FUNCTION_BLOCK T_ReleaseHandle IMPLEMENTS I_Executable
VAR
   logger : I_Logger;
	_symbolHandle : ST_SymbolHandle;
	write : T_AdsWrite;
END_VAR
VAR CONSTANT
   LOG_DEBUG : DWORD := 0;
   LOG_INFO : DWORD := ADSLOG_MSGTYPE_HINT;
   LOG_WARNING : DWORD := ADSLOG_MSGTYPE_WARN;
   LOG_ERROR : DWORD := ADSLOG_MSGTYPE_ERROR;
END_VAR

write();

PROPERTY Busy : BOOL
GET
Busy := write.Busy;
END_GET
END_PROPERTY

PROPERTY Done : BOOL
GET
Done := write.Done;
END_GET
END_PROPERTY

PROPERTY Error : BOOL
GET
Error := write.Error;
END_GET
END_PROPERTY

METHOD PRIVATE ToLog
VAR_INPUT
	Msg : STRING(255);
	LogLevel : DWORD; // generic level, can be mapped to logging framework
END_VAR
IF logger = 0 THEN
	RETURN;
	
END_IF

logger.ToLog(Msg, LogLevel);
END_METHOD

METHOD TryReleaseHandle : BOOL
VAR_INPUT
	symbolHandle : ST_SymbolHandle;
	adsTimeout : TIME := DEFAULT_ADS_TIMEOUT; // DEFAULT_ADS_TIMEOUT is T#5s;
END_VAR
VAR_OUTPUT
	status : I_Executable;
END_VAR
VAR
	readWriteOpts : ST_AdsReadWriteOptions;
END_VAR
VAR CONSTANT
	EMPTY_TARG : T_Arg;
	NO_HANDLE : DWORD := 0;
END_VAR
IF Busy THEN
	ToLog('Cannot TryReleaseHandle as Busy', LOG_WARNING);
	RETURN;
	
END_IF

_symbolHandle := symbolHandle;

readWriteOpts.AdsAddress := _symbolHandle.SymbolAddress.Ads;
readWriteOpts.IndexGroup := ADSIGRP_SYM_RELEASEHND;
readWriteOpts.IndexOffset := _symbolHandle.Handle;
readWriteOpts.WriteParams := EMPTY_TARG;
readWriteOpts.ReadParams := EMPTY_TARG;
readWriteOpts.Timeout := adsTimeout;

TryReleaseHandle := write.TryRequest( readWriteOpts, status => status );
END_METHOD

END_FUNCTION_BLOCK

(* stored: Version 1.1.0.1, ProductVersion 3.1.4024.9
   POU T_ReleaseHandle: Id {49329f98-259a-474e-af2a-fecd84d47943}, SpecialFunc None
   Property Busy: Id {96272207-f678-4a10-9cf5-b8ef46ba7d35}
   Get Get: Id {44250ed0-16f5-48a3-9001-90409046c0ef}
   Property Done: Id {7be864f6-ba4b-4200-ba89-45812d97b4f7}
   Get Get: Id {5d3e78a0-3303-486d-8b53-6242605e34a9}
   Property Error: Id {448627fd-30c5-4fab-8c29-d93ad781fa92}
   Get Get: Id {db84907b-9a03-4fc0-8191-df90268cca4d}
   Method ToLog: Id {00a93180-ffe4-4f97-a177-e40759de868d}
   Method TryReleaseHandle: Id {85758502-e02a-404f-bb25-1758ae1cc940} *)
